FUNCTION_BLOCK FB_Skill EXTENDS FB_Base IMPLEMENTS ITF_1_Skill
VAR_INPUT
	_owner: POINTER TO FB_Base;
	{attribute 'OPC.UA.DA.StructuredType':=1}
	{attribute 'OPC.UA.DA' := '1'}
	Control     : ST_SkillControl;
	{attribute 'OPC.UA.DA.StructuredType':=1}
	{attribute 'OPC.UA.DA' := '1'}
    Status      : ST_SkillStatus;
	Specific	: ST_SkillSpecific;
END_VAR
VAR_OUTPUT

END_VAR
VAR

// 	SubSkillHandler : FB_SkillHandler;
END_VAR

{warning 'Add property implementation'}
PROPERTY Busy : BOOL
GET
IF eStatus=eState.Active THEN
	Busy:=TRUE;
ELSE
	Busy:=FALSE;
END_IF
END_GET
END_PROPERTY

{attribute 'TcRpcEnable':='1'}
METHOD DeactivateSkill : BOOL
VAR_INPUT
END_VAR
Stop();
_owner^.ActivSkill:= 0;
END_METHOD

{warning 'Add property implementation'}
PROPERTY Done : BOOL
GET
Done:=bDone;
END_GET
END_PROPERTY

METHOD PROTECTED onActivate : eResult
onActivate := eResult.SUCCESS;
      RETURN;
      // ---- Init ----
_transitionresult:=eResult.None;



// ---- Change ----




// ---- Check ----
_transitionresult := eResult.SUCCESS;


// ---- Change State ----
IF _transitionresult= eResult.SUCCESS THEN
	State:=eState.Active;
ELSIF _transitionresult= eResult.FAILURE THEN
	State:=eState.Inactive;
ELSIF _transitionresult= eResult.ERROR THEN
	State:=eState.ErrorProcessing;
ELSE
	ADSLOGSTR(ADSLOG_MSGTYPE_WARN,'Transitionresult from onActivate is None','');
END_IF
END_METHOD

METHOD PROTECTED onCleanup : eResult
onCleanup := eResult.SUCCESS;
      RETURN;
      // ---- Init ----
_transitionresult:=eResult.None;



// ---- Change ----



// ---- Check ----
_transitionresult := eResult.SUCCESS;


// ---- Change State ----
IF _transitionresult= eResult.SUCCESS THEN
	State:=eState.Unconfigured;
ELSIF _transitionresult= eResult.FAILURE THEN
	ADSLOGSTR(ADSLOG_MSGTYPE_WARN,'Transitionresult from onCleanup is FAILURE ','');
ELSIF _transitionresult= eResult.ERROR THEN
	State:=eState.ErrorProcessing;
ELSE
	ADSLOGSTR(ADSLOG_MSGTYPE_WARN,'Transitionresult from onCleanup is NONE','');
END_IF
END_METHOD

METHOD PROTECTED onConfigure : eResult
onConfigure := eResult.SUCCESS;
      RETURN;
      // ---- Init ----
_transitionresult:=eResult.None;



// ---- Change ----


// ---- Check ----
_transitionresult := eResult.SUCCESS;


// ---- Change State ----
IF _transitionresult= eResult.SUCCESS THEN
	State:=eState.Inactive;
ELSIF _transitionresult= eResult.FAILURE THEN
	State:=eState.Unconfigured;
ELSIF _transitionresult= eResult.ERROR THEN
	State:=eState.ErrorProcessing;
ELSE
	ADSLOGSTR(ADSLOG_MSGTYPE_WARN,'Transitionresult from onConfigure is None','');
END_IF
END_METHOD

METHOD PROTECTED onDeactivate : eResult
onDeactivate := eResult.SUCCESS;
      RETURN;
      // ---- Init ----
_transitionresult:=eResult.None;



// ---- Change ----
 //Stopping SFC



// ---- Check ----
_transitionresult := eResult.SUCCESS;


// ---- Change State ----
IF _transitionresult= eResult.SUCCESS THEN
	State:=eState.Inactive;
ELSIF _transitionresult= eResult.FAILURE THEN
	ADSLOGSTR(ADSLOG_MSGTYPE_WARN,'Transitionresult from onDeactivate is FAILURE','');
ELSIF _transitionresult= eResult.ERROR THEN
	State:=eState.ErrorProcessing;
ELSE
	ADSLOGSTR(ADSLOG_MSGTYPE_WARN,'Transitionresult from onDeactivate is None','');
END_IF
END_METHOD

METHOD PROTECTED onError : eResult
onError := eResult.SUCCESS;
      RETURN;
      // ---- Init ----
_transitionresult:=eResult.None;



// ---- Change ----





// ---- Check ----
_transitionresult := eResult.SUCCESS;


// ---- Change State ----
IF _transitionresult= eResult.SUCCESS THEN
	State:=eState.Unconfigured;
ELSIF _transitionresult= eResult.FAILURE THEN
	State:=eState.Finalized;
ELSIF _transitionresult= eResult.ERROR THEN
	ADSLOGSTR(ADSLOG_MSGTYPE_WARN,'Transitionresult from onError is Error','');
ELSE
	ADSLOGSTR(ADSLOG_MSGTYPE_WARN,'Transitionresult from onError is None','');
END_IF
END_METHOD

METHOD PROTECTED onShutdown : eResult
onShutdown := eResult.SUCCESS;
      RETURN;
      // ---- Init ----
_transitionresult:=eResult.None;



// ---- Change ----



// ---- Check ----
_transitionresult := eResult.SUCCESS;


// ---- Change State ----
IF _transitionresult= eResult.SUCCESS THEN
	State:=eState.Finalized;
ELSIF _transitionresult= eResult.FAILURE THEN
	ADSLOGSTR(ADSLOG_MSGTYPE_WARN,'Transitionresult from onShutdown is FAILURE','');
ELSIF _transitionresult= eResult.ERROR THEN
	State:=eState.ErrorProcessing;
ELSE
	ADSLOGSTR(ADSLOG_MSGTYPE_WARN,'Transitionresult from onShutdown is None','');
END_IF
END_METHOD

{warning 'Add method implementation '}
METHOD INTERNAL Pause : BOOL
IF eStatus=eState.Active THEN
	SFCPause:=TRUE;
END_IF
END_METHOD

{warning 'Add method implementation '}
METHOD INTERNAL Restart : BOOL //Stay activ, but restart
SFCReset:=True;
END_METHOD

{warning 'Add method implementation '}
METHOD INTERNAL Resume : BOOL
SFCPause:=False;
END_METHOD

{warning 'Add method implementation '}
METHOD INTERNAL Start : BOOL

VAR
	config_succ: BOOL:=TRUE;
	act_succ: BOOL;
END_VAR
IF State = eState.Unconfigured THEN
	config_succ:=FALSE;
	config_succ := Configure();
	ADSLOGSTR(
    msgCtrlMask := ADSLOG_MSGTYPE_HINT,
    msgFmtStr   := 'Autoconfiguring Skill %s because Start was called an State = unconfigured',
    strArg      := Path
);
END_IF
IF config_succ THEN
	act_succ := Activate();
END_IF


IF act_succ THEN 
	Start:=TRUE; 
	ADSLOGSTR(
    msgCtrlMask := ADSLOG_MSGTYPE_HINT,
    msgFmtStr   := 'Starting Skill: %s',
    strArg      := Name
);
 END_IF
END_METHOD

{attribute 'TcRpcEnable':='1'}
METHOD StartSkill
VAR_INPUT
// 	pSkill : POINTER TO FB_SKILL;
// 	name: STRING := '';
END_VAR

VAR
	toolready: BOOL;
	i: INT;
END_VAR
Start();
_owner^.ActivSkill:= THIS;


// IF name<>'' THEN
// 	FOR i := TO_INT(LOWER_BOUND(_owner^.pA_Skills, 1)) TO TO_INT(UPPER_BOUND(_owner^.pA_Skills, 1)) DO
// 		IF _owner^.pA_Skills[i]<>0 THEN
// 			IF FIND(STR1:=pA_Skills[i]^.Name, STR2:=name)<>0 THEN
// 				pSkill:=_owner^.pA_Skills[i];
// 				ADSLOGSTR(
// 					msgCtrlMask := ADSLOG_MSGTYPE_HINT,
// 					msgFmtStr   := 'CallSkill: Found by name: %s',
// 					strArg      := _owner^.pA_Skills[i]^.Name
// 				);
// 				EXIT;
// 			END_IF
// 		END_IF
// 	END_FOR
// 	
// END_IF
// 
// 
// IF pSkill<>0 THEN
// 	activSkill:= pSkill;
// 	
// // 	toolready:=TRUE;
// // 	IF _owner^.pTool<>0 THEN
// // 		toolready:=FALSE;
// // 		IF _owner^.pTool^.State = eState.Active THEN
// // 			toolready:=TRUE;
// // 		END_IF
// // 	END_IF
// 	
// 	
// 	pSkill^.Start();
// ELSE
// 	ADSLOGSTR(
//     msgCtrlMask := ADSLOG_MSGTYPE_ERROR,
//     msgFmtStr   := 'CallSkill: Pointer to Skill is empty: %s',
//     strArg      := _owner^.Path
// );
// END_IF
END_METHOD

{warning 'Add method implementation '}
METHOD INTERNAL Stop : BOOL
IF eStatus=eState.Active THEN
	SFCPause:=TRUE;
	super^.Deactivate();
END_IF
END_METHOD

END_FUNCTION_BLOCK

(* stored: Version 1.1.0.1, ProductVersion 3.1.4026.18
   POU FB_Skill: Id {de568c3b-e8e2-4fe8-b2d6-5e89933abc51}, SpecialFunc None
   Folder Internal: Id {20bd2501-e1eb-4995-8337-668ddeba1c4c}
   Folder Public: Id {242a8bf6-3dc5-446b-a89d-936e418b8756}
   Folder StateControl: Id {31a6bbdd-3ba2-4185-a10e-7900c7f6f8d3}
   Property Busy: Id {59c0b902-0e96-4aa6-80c4-17e0cd6c8a94}
   Get Get: Id {f0fed57d-7011-4c26-a36d-51ead2ced228}
   Method DeactivateSkill: Id {10338084-d473-478a-aa27-fc35b9873599}
   Property Done: Id {d7794fd0-d52a-411f-ae53-4abe695b2781}
   Get Get: Id {a38fbf64-c78a-4e85-9631-248ee16d04de}
   Method onActivate: Id {ecc4deb5-0154-49af-a556-dd604d8dfee8}
   Method onCleanup: Id {39f97e2b-ba11-4e41-adb8-2fa35d8f889b}
   Method onConfigure: Id {017eb5d1-e54b-4d70-a6cb-15146fd5331d}
   Method onDeactivate: Id {0937e09f-333a-4e3a-844b-9f0a153fa24d}
   Method onError: Id {5ea8935e-cd95-4d1d-b64a-37648a2cf45e}
   Method onShutdown: Id {f185d0d9-18df-4a16-be3c-0516eebae000}
   Method Pause: Id {14cdbcfb-a616-4591-a925-297ff9db8a79}
   Method Restart: Id {fd5f86ff-0d6c-49e6-bddb-d9209e3aabfc}
   Method Resume: Id {3f8922d2-b958-4616-a24f-75320fdcbb9f}
   Method Start: Id {ccb135ee-6087-41f8-8be8-8d6e596b5080}
   Method StartSkill: Id {d8fc5668-9fa7-43c2-a944-aada2bd4cb8c}
   Method Stop: Id {4c723123-1adf-4d21-9269-2419097dc023} *)
